(* IEC 61131-3 sources: ArfBotOS/Codesys-4/ArfBotOS.fbsdev/Application.iecapp^/FUN/cnc/FB_CncPathPlanner.fb.st^, 4 files *)

(* ---- M_Execute.meth.st ---- *)
METHOD PUBLIC M_Execute : BOOL
VAR_INPUT
	Filename: STRING := 'CNC_FromFile.cnc';
END_VAR

_Filename := CONCAT(_BaseCncDirectory, Filename);
_Execute:=TRUE;
Done := FALSE;
END_METHOD

(* ---- M_Reset.meth.st ---- *)
METHOD PUBLIC M_Reset : BOOL
VAR_INPUT
END_VAR

_Reset := TRUE;
Error := FALSE;
ErrorDescription := '';
END_METHOD

(* ---- M_SetOriConvention.meth.st ---- *)
METHOD PUBLIC M_SetOriConvention : BOOL
VAR_INPUT
	OriConvention: SMC_ORI_CONVENTION := SMC_ORI_CONVENTION.ZYZ;
END_VAR

_OriConvention := OriConvention;
GVL_App.OriConvention := OriConvention;
END_METHOD

(* ---- M_SetStartPosition.meth.st ---- *)
METHOD PUBLIC M_SetStartPosition : BOOL
VAR_INPUT
	StartPos: SMC_PosInfo;
END_VAR

_StartPos := StartPos;
END_METHOD
